FUNCTION_BLOCK FB_PlantControl
VAR_INPUT
	Auto_In : BOOL;
	Manual_In : BOOL;
	
	Start_In : BOOL;
	Stop_In : BOOL;
	Reset_In : BOOL;
	
	EmgStop_In : BOOL;
	
END_VAR
VAR_OUTPUT
	Auto_Out : BOOL;
	Manual_Out : BOOL;
	
	Startet_Out : BOOL;
	Stopped_Out : BOOL;
	Reset_Out : BOOL;
	ResetEmgStop_Out_5s :BOOL;
	
	EmgStopped_Out : BOOL;
END_VAR
VAR
END_VAR
VAR_IN_OUT
	Ctrl_Plant : Udt_PlantControl_Out;
END_VAR

VAR CONSTANT
	SR_Auto: SR;
	SR_Man : SR;
	
	SR_start : SR;
	SR_Stop : SR;
	
	EmgResetTimerOff : Tc2_Standard.TON;
END_VAR

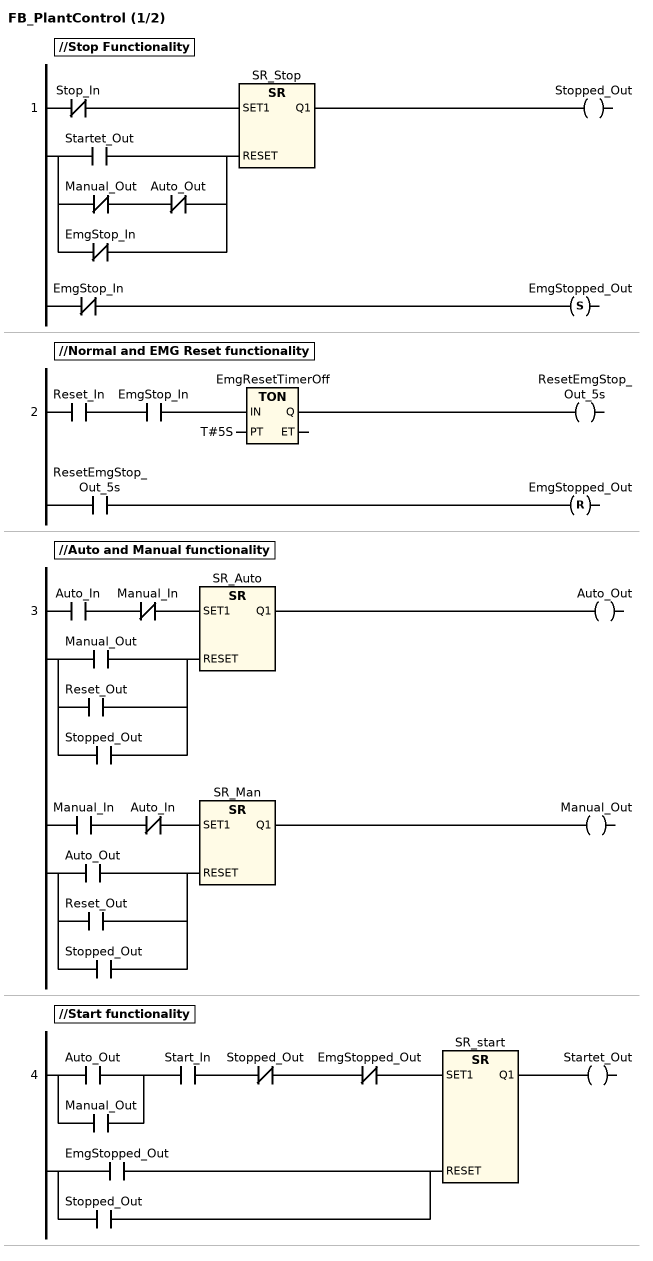
// NETWORK 1
// label: //Stop Functionality
SR_Stop(SET1 := NOT Stop_In, RESET := Startet_Out OR NOT Manual_Out AND NOT Auto_Out OR NOT EmgStop_In); // SR
Stopped_Out := SR_Stop.Q1;
EmgStopped_Out S= NOT EmgStop_In;

// NETWORK 2
// label: //Normal and EMG Reset functionality
EmgResetTimerOff(IN := Reset_In AND EmgStop_In, PT := T#5S); // TON
ResetEmgStop_Out_5s := EmgResetTimerOff.Q;
EmgStopped_Out R= ResetEmgStop_Out_5s;

// NETWORK 3
// label: //Auto and Manual functionality
SR_Auto(SET1 := Auto_In AND NOT Manual_In, RESET := Manual_Out OR Reset_Out OR Stopped_Out); // SR
Auto_Out := SR_Auto.Q1;
SR_Man(SET1 := Manual_In AND NOT Auto_In, RESET := Auto_Out OR Reset_Out OR Stopped_Out); // SR
Manual_Out := SR_Man.Q1;

// NETWORK 4
// label: //Start functionality
SR_start(SET1 := (Auto_Out OR Manual_Out) AND Start_In AND NOT Stopped_Out AND NOT EmgStopped_Out, RESET := EmgStopped_Out OR Stopped_Out); // SR
Startet_Out := SR_start.Q1;

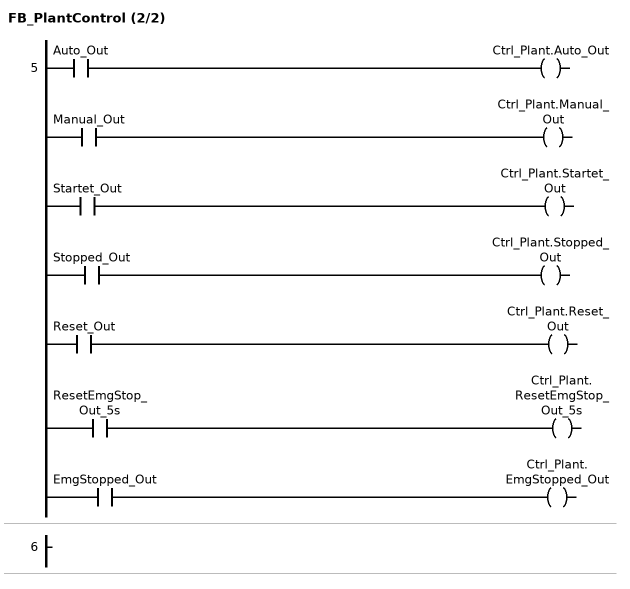
// NETWORK 5
Ctrl_Plant.Auto_Out := Auto_Out;
Ctrl_Plant.Manual_Out := Manual_Out;
Ctrl_Plant.Startet_Out := Startet_Out;
Ctrl_Plant.Stopped_Out := Stopped_Out;
Ctrl_Plant.Reset_Out := Reset_Out;
Ctrl_Plant.ResetEmgStop_Out_5s := ResetEmgStop_Out_5s;
Ctrl_Plant.EmgStopped_Out := EmgStopped_Out;

// NETWORK 6

END_FUNCTION_BLOCK

(* stored: Version 1.1.0.1, ProductVersion 3.1.4024.13
   POU FB_PlantControl: Id {b53adaf6-8506-476c-8298-f670f349374b}, SpecialFunc None *)
